// TIA Portal V17 export
// export: Created 2025-06-25T13:13:27.6865455Z, ExportSetting WithDefaults, DisplayName Totally Integrated Automation Portal, DisplayVersion V17 Update 8, DisplayName TIA Portal Openness, DisplayVersion V17 Update 8, DisplayName TIA Portal Version Control Interface, DisplayVersion V17, DisplayName STEP 7 Professional, DisplayVersion V17 Update 8, DisplayName STEP 7 Safety, DisplayVersion V17 Update 6, DisplayName WinCC Advanced, DisplayVersion V17 Update 8
TYPE "stDeviationAlarm"
// stored: IsFailsafeCompliant false
   STRUCT
      bEnable : Bool := true;   // 1 = enable, 0 = block
      fDeviationLimit : Real;   // Alarm threshold
      tActivationDelay : Time;   // Alarm activation delay
      sState : "stAlarmState";   // Alarm
   END_STRUCT;
END_TYPE
